ABB RAPID module: Wobj_DANinclindo.mod

MODULE Wobj_DANinclindo
	! Points are read in order of declaration.
  ! Please do not change the order of points!

  LOCAL PERS robtarget pWobj_O_PointX1:=[[366.1427,617.3132,205.8221],[0.207270815968513,-0.196583494544029,0.934262812137604,0.213416919112206],[0,0,0,0],[9E+09,9E+09,9E+09,9E+09,9E+09,9E+09]];
	LOCAL PERS robtarget pWobj_O_PointX2:=[[364.9155,431.0839,8.512452],[0.207275673747063,-0.196578025817871,0.934265732765198,0.213404342532158],[0,1,-2,0],[9E+09,9E+09,9E+09,9E+09,9E+09,9E+09]];
	LOCAL PERS robtarget pWobj_O_PointY1:=[[81.87099,617.6058,194.193],[0.207271575927734,-0.196583420038223,0.934262573719025,0.213417321443558],[0,-1,1,0],[9E+09,9E+09,9E+09,9E+09,9E+09,9E+09]];

ENDMODULE
